Staubli VAL3: Control_LeftS.pgx

public program Control_LeftS(string x_sLeftList)
  local bool l_bRes
  local string l_sBuff[20]
begin

  call Str_SplitComma(l_bRes,x_sLeftList,l_sBuff)
  if !l_bRes
    return
  endIf

call Control_Left(l_sBuff)
end
